{attribute 'linkalways'} 
{attribute 'no_explicit_call' := 'This FB is a CLASS and must be accessed using methods or properties'}
{attribute 'enable_dynamic_creation'}
FUNCTION_BLOCK FINAL MAX_WORD EXTENDS Node
VAR
	in1 : _WORD(0);
	in2 : _WORD(0);
	out : _WORD(0);
END_VAR

METHOD PUBLIC Clone : I_Node
VAR
	pNode : POINTER TO MAX_WORD;
END_VAR
pNode := __NEW(MAX_WORD);
Clone := pNode^;
END_METHOD

METHOD FB_init : BOOL
VAR_INPUT
	bInitRetains : BOOL; // if TRUE, the retain variables are initialized (warm start / cold start)
	bInCopyCode : BOOL;  // if TRUE, the instance afterwards gets moved into the copy code (online change)
END_VAR
AddInput('in1',THIS^.in1);
AddInput('in2',THIS^.in2);
AddOutput('out', THIS^.out);
END_METHOD

METHOD PROTECTED OnExecute
VAR
END_VAR
out.Value := MAX(in1.Value, in2.Value);
END_METHOD

END_FUNCTION_BLOCK

(* stored: Version 1.1.0.1, ProductVersion 3.1.4024.15
   POU MAX_WORD: Id {5eed6fd2-1740-4b6c-9c12-7f69d705cf0c}, SpecialFunc None
   Folder Constructor: Id {ab336714-f912-44b8-ad81-e746475c8e73}
   Method Clone: Id {2d845f36-67ab-4351-b49b-c10c6ab83064}
   Method FB_init: Id {23e5f73c-593b-48dc-bf5c-84294f6f66f8}
   Method OnExecute: Id {297986e7-aab4-4de9-a05b-ce5133ef4651} *)
